// Mitsubishi GX Works2 project: 2023-06-27 #2 생산자동화기능사 10번   PLC: Q03UDV
// 생산자동화기능사

// global labels: Global1
VAR_GLOBAL
  PB1 AT X0 : BOOL;
  PB2 AT X1 : BOOL;
  정지 AT X2 : BOOL;
  공급후진 AT X3 : BOOL;
  공급전진 AT X4 : BOOL;
  가공후진 AT X5 : BOOL;
  가공전진 AT X6 : BOOL;
  송출후진 AT X7 : BOOL;
  송출전진 AT X8 : BOOL;
  배출후진 AT X9 : BOOL;
  배출전진 AT X0A : BOOL;
  매거진 AT X0B : BOOL;
  금속센서 AT X0F : BOOL;
  PB3 AT X10 : BOOL;
  적색 AT Y20 : BOOL;
  황색 AT Y21 : BOOL;
  녹색 AT Y22 : BOOL;
  공급1 AT Y23 : BOOL;
  공급2 AT Y24 : BOOL;
  가공 AT Y25 : BOOL;
  드릴 AT Y26 : BOOL;
  송출 AT Y27 : BOOL;
  배출 AT Y28 : BOOL;
  컨베이어 AT Y29 : BOOL;
END_VAR

PROGRAM 테스트동작
VAR
  PHASE : INT;
END_VAR
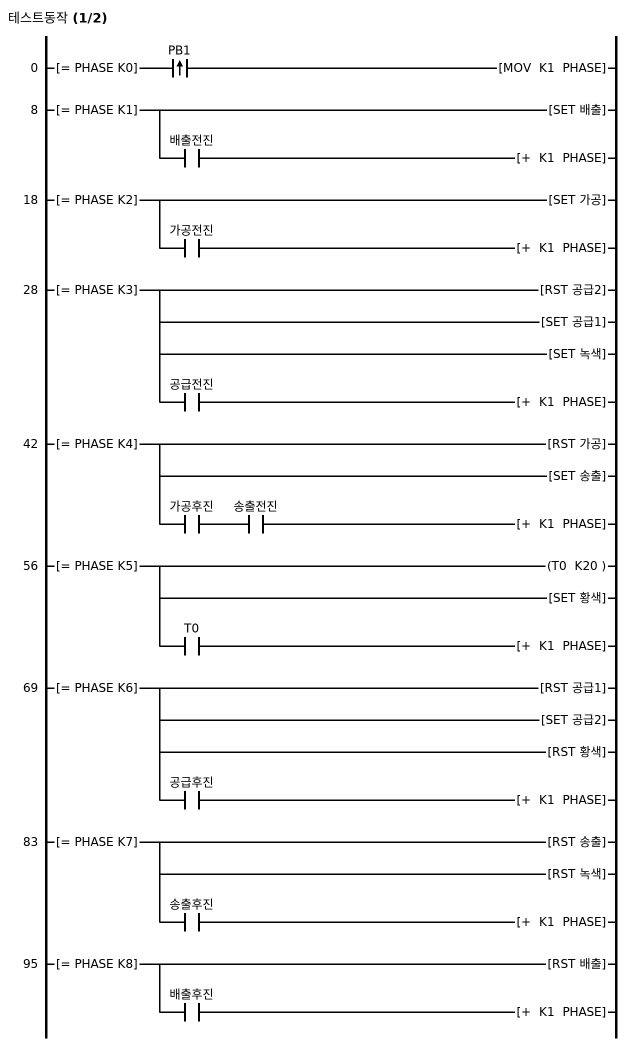
0     LD=     PHASE K0
      ANDP    PB1
      MOV     K1 PHASE
8     LD=     PHASE K1
      SET     배출
      AND     배출전진
      +       K1 PHASE
18    LD=     PHASE K2
      SET     가공
      AND     가공전진
      +       K1 PHASE
28    LD=     PHASE K3
      RST     공급2
      SET     공급1
      SET     녹색
      AND     공급전진
      +       K1 PHASE
42    LD=     PHASE K4
      RST     가공
      SET     송출
      AND     가공후진
      AND     송출전진
      +       K1 PHASE
56    LD=     PHASE K5
      OUT     T0 K20
      SET     황색
      AND     T0
      +       K1 PHASE
69    LD=     PHASE K6
      RST     공급1
      SET     공급2
      RST     황색
      AND     공급후진
      +       K1 PHASE
83    LD=     PHASE K7
      RST     송출
      RST     녹색
      AND     송출후진
      +       K1 PHASE
95    LD=     PHASE K8
      RST     배출
      AND     배출후진
      +       K1 PHASE
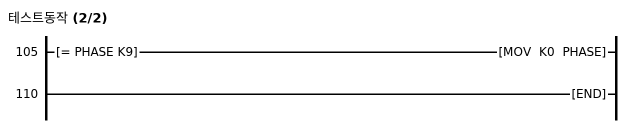
105   LD=     PHASE K9
      MOV     K0 PHASE
110   END
END_PROGRAM

PROGRAM 단속및연속동작
VAR
  PHASE : INT;
  MODE : INT;
END_VAR
VAR CONSTANT
  단속 : INT;
  연속 : INT := 1;
END_VAR
VAR
  STORAGE : INT;
  METAL : INT;
END_VAR
VAR CONSTANT
  금속 : INT := 1;
  비금속 : INT := 2;
END_VAR
VAR
  BLINK : ARRAY [0..7] OF BOOL;
  EMG : INT;
  PHASE1 : INT;
  드릴1 : BOOL;
  컨베이어1 : BOOL;
  녹색1 : BOOL;
  황색1 : BOOL;
END_VAR
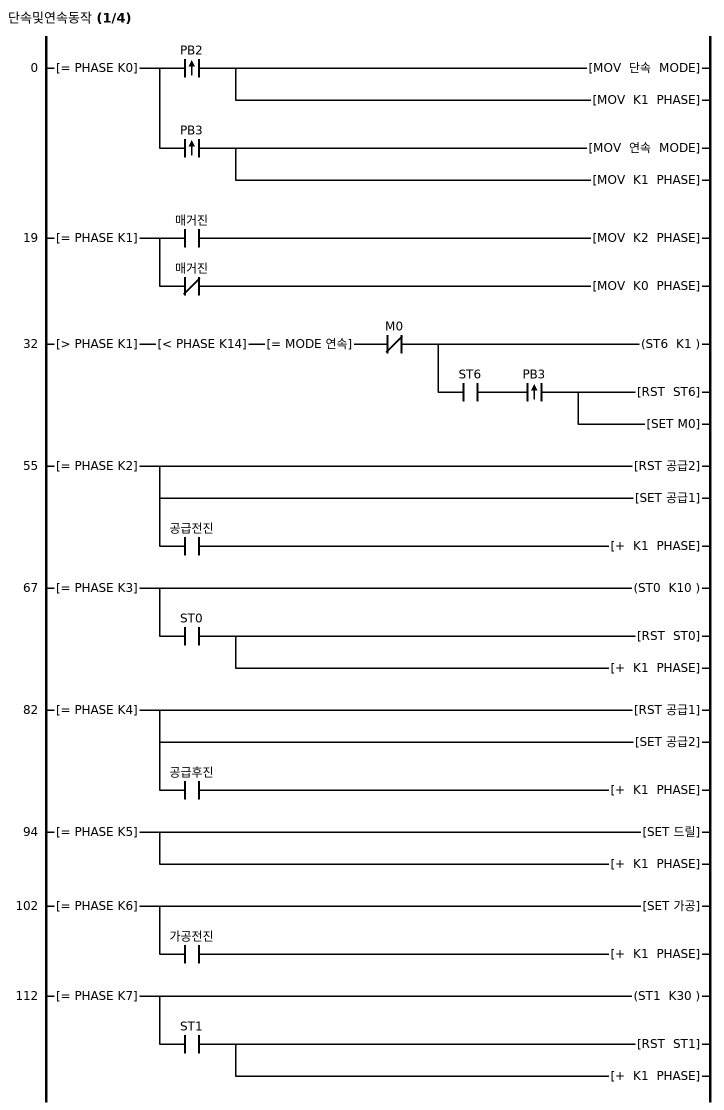
0     LD=     PHASE K0
      MPS
      ANDP    PB2
      MOV     단속 MODE
      MOV     K1 PHASE
      MPP
      ANDP    PB3
      MOV     연속 MODE
      MOV     K1 PHASE
19    LD=     PHASE K1
      MPS
      AND     매거진
      MOV     K2 PHASE
      MPP
      ANI     매거진
      MOV     K0 PHASE
32    LD>     PHASE K1
      AND<    PHASE K14
      AND=    MODE 연속
      ANI     M0
      OUT     ST6 K1
      AND     ST6
      ANDP    PB3
      RST     ST6
      SET     M0
55    LD=     PHASE K2
      RST     공급2
      SET     공급1
      AND     공급전진
      +       K1 PHASE
67    LD=     PHASE K3
      OUT     ST0 K10
      AND     ST0
      RST     ST0
      +       K1 PHASE
82    LD=     PHASE K4
      RST     공급1
      SET     공급2
      AND     공급후진
      +       K1 PHASE
94    LD=     PHASE K5
      SET     드릴
      +       K1 PHASE
102   LD=     PHASE K6
      SET     가공
      AND     가공전진
      +       K1 PHASE
112   LD=     PHASE K7
      OUT     ST1 K30
      AND     ST1
      RST     ST1
      +       K1 PHASE
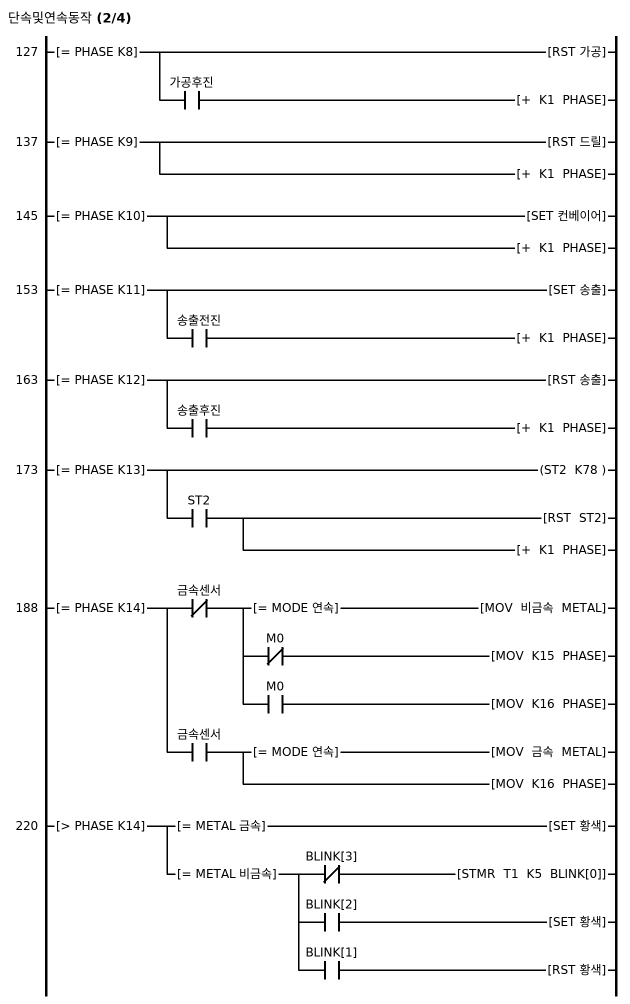
127   LD=     PHASE K8
      RST     가공
      AND     가공후진
      +       K1 PHASE
137   LD=     PHASE K9
      RST     드릴
      +       K1 PHASE
145   LD=     PHASE K10
      SET     컨베이어
      +       K1 PHASE
153   LD=     PHASE K11
      SET     송출
      AND     송출전진
      +       K1 PHASE
163   LD=     PHASE K12
      RST     송출
      AND     송출후진
      +       K1 PHASE
173   LD=     PHASE K13
      OUT     ST2 K78
      AND     ST2
      RST     ST2
      +       K1 PHASE
188   LD=     PHASE K14
      MPS
      ANI     금속센서
      MPS
      AND=    MODE 연속
      MOV     비금속 METAL
      MRD
      ANI     M0
      MOV     K15 PHASE
      MPP
      AND     M0
      MOV     K16 PHASE
      MPP
      AND     금속센서
      MPS
      AND=    MODE 연속
      MOV     금속 METAL
      MPP
      MOV     K16 PHASE
220   LD>     PHASE K14
      MPS
      AND=    METAL 금속
      SET     황색
      MPP
      AND=    METAL 비금속
      MPS
      ANI     BLINK[3]
      STMR    T1 K5 BLINK[0]
      MRD
      AND     BLINK[2]
      SET     황색
      MPP
      AND     BLINK[1]
      RST     황색
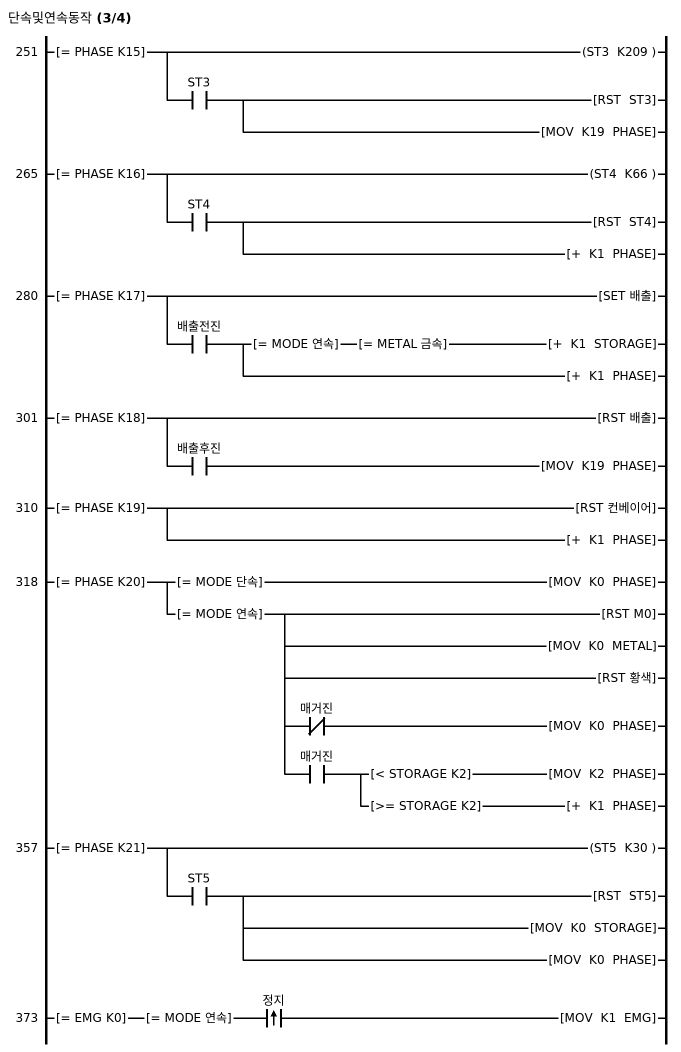
251   LD=     PHASE K15
      OUT     ST3 K209
      AND     ST3
      RST     ST3
      MOV     K19 PHASE
265   LD=     PHASE K16
      OUT     ST4 K66
      AND     ST4
      RST     ST4
      +       K1 PHASE
280   LD=     PHASE K17
      SET     배출
      AND     배출전진
      MPS
      AND=    MODE 연속
      AND=    METAL 금속
      +       K1 STORAGE
      MPP
      +       K1 PHASE
301   LD=     PHASE K18
      RST     배출
      AND     배출후진
      MOV     K19 PHASE
310   LD=     PHASE K19
      RST     컨베이어
      +       K1 PHASE
318   LD=     PHASE K20
      MPS
      AND=    MODE 단속
      MOV     K0 PHASE
      MPP
      AND=    MODE 연속
      RST     M0
      MOV     K0 METAL
      RST     황색
      MPS
      ANI     매거진
      MOV     K0 PHASE
      MPP
      AND     매거진
      MPS
      AND<    STORAGE K2
      MOV     K2 PHASE
      MPP
      AND>=   STORAGE K2
      +       K1 PHASE
357   LD=     PHASE K21
      OUT     ST5 K30
      AND     ST5
      RST     ST5
      MOV     K0 STORAGE
      MOV     K0 PHASE
373   LD=     EMG K0
      AND=    MODE 연속
      ANDP    정지
      MOV     K1 EMG
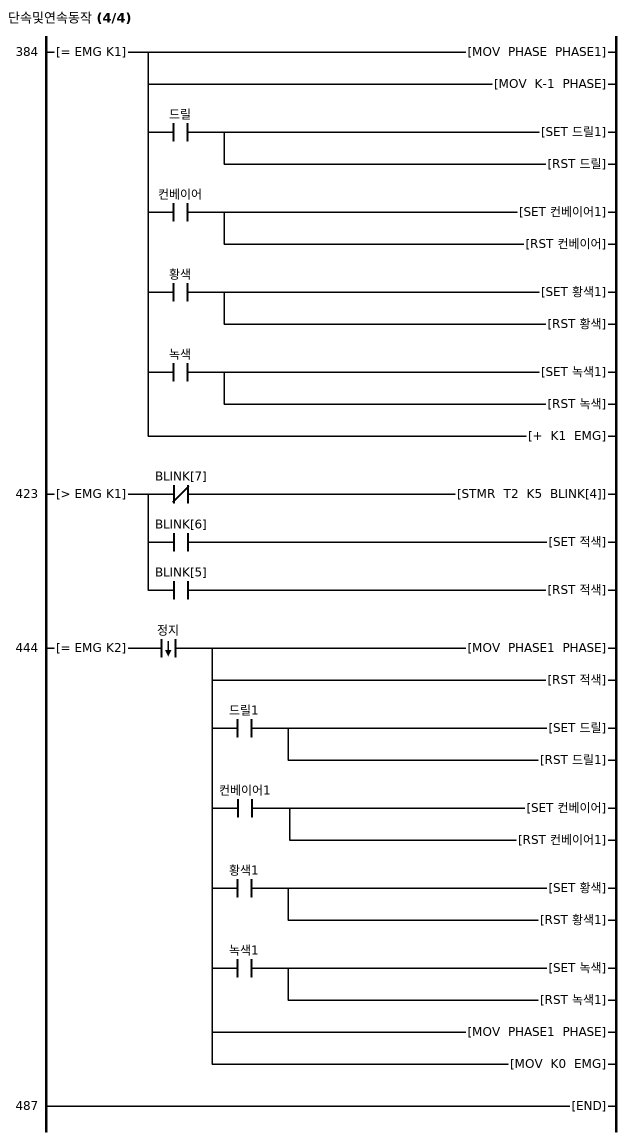
384   LD=     EMG K1
      MOV     PHASE PHASE1
      MOV     K-1 PHASE
      MPS
      AND     드릴
      SET     드릴1
      RST     드릴
      MRD
      AND     컨베이어
      SET     컨베이어1
      RST     컨베이어
      MRD
      AND     황색
      SET     황색1
      RST     황색
      MRD
      AND     녹색
      SET     녹색1
      RST     녹색
      MPP
      +       K1 EMG
423   LD>     EMG K1
      MPS
      ANI     BLINK[7]
      STMR    T2 K5 BLINK[4]
      MRD
      AND     BLINK[6]
      SET     적색
      MPP
      AND     BLINK[5]
      RST     적색
444   LD=     EMG K2
      ANDF    정지
      MOV     PHASE1 PHASE
      RST     적색
      MPS
      AND     드릴1
      SET     드릴
      RST     드릴1
      MRD
      AND     컨베이어1
      SET     컨베이어
      RST     컨베이어1
      MRD
      AND     황색1
      SET     황색
      RST     황색1
      MRD
      AND     녹색1
      SET     녹색
      RST     녹색1
      MPP
      MOV     PHASE1 PHASE
      MOV     K0 EMG
487   END
END_PROGRAM
